Staubli VAL3: test.pjx

--- test.pjx ---
Parameters version=s7.8.3 stackSize=5000 millimeterUnit=true
Program file=start.pgx
Program file=stop.pgx
Data file=test.dtx

--- test.dtx ---
mdesc mNomSpeed
string sTarget{}
  [Key1] = {}
string sOrig{}
  [Key1] = {}
  [Key2] = {}
  [Key3] = {}
  [Key4] = {}
  [Key5] = {}
  [Key6] = {}
  [Key7] = {}
  [Key8] = {}
  [Key9] = {}
  [Key10] = {}
string sKey

--- start.pgx ---
program start()
  local string l_sKey
begin
  while size(sOrig)>8
    l_sKey=first(sOrig)
    delete(sOrig[l_sKey])
  endWhile

//  if first(sOrig)==""
//    delete(sTarget["Key1"])
//    popUpMsg("空")
//  else
//    popUpMsg(toString("",size(sOrig)))
//  endIf


   // popUpMsg(toString("",size(sTarget)))


end
